(* IEC 61131-3 sources: SmartHomeNew/snapshots/2026-05-05 (part 2) *)

(* ---- PRG_IO_Write.st ---- *)
PROGRAM PRG_IO_Write
VAR
    L_i : INT;
    L_Heating_Forced_Off : BOOL;
    L_Vent_Forced_Off : BOOL;
    L_Water_Forced_Off : BOOL;
    L_Access_Forced_Off : BOOL;
    L_Access_Safety_Override : BOOL;
    L_Global_Hard_Stop : BOOL;
    L_Gas_Safety_Stop : BOOL;
    L_Freeze_Active : BOOL;
    L_Gas_Fire_Siren_Enable : BOOL;
    fbTrace : FB_Trace_Write;
END_VAR

L_Global_Hard_Stop := GVL_COMMAND_SHADOW.G_Heating_Emergency_Stop;
L_Gas_Safety_Stop := GVL_COMMAND_SHADOW.G_Heating_Gas_Safety_Stop OR GVL_COMMAND_SHADOW.G_Boiler_Stop;
L_Freeze_Active := GVL_STATE.G_Safety_Freeze_Risk;
L_Gas_Fire_Siren_Enable := GVL_ALARM.G_Gas_Fire_Siren OR GVL_ALARM.G_Global_Siren OR GVL_ALARM.G_Global_Critical;

IF NOT GVL_STATUS.G_Is_Active_PLC OR L_Global_Hard_Stop THEN
    FOR L_i := 1 TO GVL_CONSTANTS.C_MAX_HEATING_CIRCUITS DO GVL_IO.DO_Zone_Valves[L_i] := FALSE; END_FOR;
    FOR L_i := 1 TO GVL_CONSTANTS.C_MAX_MANIFOLDS DO GVL_IO.DO_Manifold_Pumps[L_i] := FALSE; GVL_IO.AO_Manifold_Valves[L_i] := 0; END_FOR;
    GVL_IO.DO_DHW_Heating_Pump := FALSE;
    GVL_IO.DO_DHW_Circ_Pump := FALSE;
    GVL_IO.DO_Backup_Circulation_Pump := FALSE;
    GVL_IO.DO_Electric_Heater_Enable := FALSE;
    FOR L_i := 1 TO GVL_CONSTANTS.C_MAX_SUPPLY_FANS DO GVL_IO.AO_Supply_Fans[L_i] := 0; END_FOR;
    FOR L_i := 1 TO GVL_CONSTANTS.C_MAX_EXHAUST_FANS DO GVL_IO.AO_Exhaust_Fans[L_i] := 0; END_FOR;
    FOR L_i := 1 TO GVL_CONSTANTS.C_MAX_WATER_ZONES DO GVL_IO.DO_Water_Zone_Enable[L_i] := FALSE; END_FOR;
    FOR L_i := 1 TO GVL_CONSTANTS.C_MAX_LIGHT_ZONES DO GVL_IO.AO_Lighting_Levels[L_i] := 0; END_FOR;
    FOR L_i := 1 TO GVL_CONSTANTS.C_MAX_BLINDS DO GVL_IO.AO_Blinds_Positions[L_i] := 1000; END_FOR;
    FOR L_i := 1 TO GVL_CONSTANTS.C_MAX_SOCKETS DO GVL_IO.DO_Sockets[L_i] := FALSE; END_FOR;
    GVL_IO.DO_Gate_Open := FALSE;
    GVL_IO.DO_Wicket_Open := FALSE;
    GVL_IO.DO_Lock_1_Open := FALSE;
    GVL_IO.DO_Lock_1_Close := FALSE;
    GVL_IO.DO_Lock_2_Open := FALSE;
    GVL_IO.DO_Lock_2_Close := FALSE;
    GVL_IO.DO_Gas_Siren := L_Gas_Fire_Siren_Enable AND GVL_ALARM.G_Gas_Alarm_Active;
    GVL_IO.DO_Fire_Siren := L_Gas_Fire_Siren_Enable AND GVL_ALARM.G_Fire_Alarm_Active;
    GVL_IO.DO_Security_Siren := GVL_ALARM.G_Security_Siren OR (GVL_ALARM.G_Global_Siren AND GVL_ALARM.G_Security_Alarm);
    GVL_IO.DO_Gas_Valve_Close := TRUE;
    RETURN;
END_IF;

L_Heating_Forced_Off := GVL_COMMAND_SHADOW.G_Heating_Block;
L_Vent_Forced_Off := GVL_COMMAND_SHADOW.G_Vent_Stop OR GVL_COMMAND_SHADOW.G_Vent_Block;
L_Water_Forced_Off := GVL_COMMAND_SHADOW.G_Water_Block OR GVL_COMMAND_SHADOW.G_Water_Emergency_Stop;

L_Access_Safety_Override := (GVL_SAFETY_SHUTDOWN.G_Safety_Mode = FIRE) OR (GVL_SAFETY_SHUTDOWN.G_Safety_Mode = GAS);
L_Access_Forced_Off := GVL_SAFETY_RECOVERY.G_Recovery_Active AND NOT L_Access_Safety_Override;

FOR L_i := 1 TO GVL_CONSTANTS.C_MAX_HEATING_CIRCUITS DO
    IF (L_i > GVL_SYSTEM_SIZE_CONFIG.G_Active_Heating_Circuits) OR L_Heating_Forced_Off THEN
        GVL_IO.DO_Zone_Valves[L_i] := FALSE;
    ELSE
        GVL_IO.DO_Zone_Valves[L_i] := GVL_HEATING_OUTPUT.DO_Zone_Valves[L_i];
    END_IF;
END_FOR;

FOR L_i := 1 TO GVL_CONSTANTS.C_MAX_MANIFOLDS DO
    IF L_Heating_Forced_Off AND NOT (L_Gas_Safety_Stop AND L_Freeze_Active) THEN
        GVL_IO.DO_Manifold_Pumps[L_i] := FALSE;
        GVL_IO.AO_Manifold_Valves[L_i] := 0;
    ELSE
        GVL_IO.DO_Manifold_Pumps[L_i] := GVL_HEATING_OUTPUT.DO_Manifold_Pumps[L_i];
        GVL_IO.AO_Manifold_Valves[L_i] := GVL_HEATING_OUTPUT.AO_Manifold_Valves[L_i];
    END_IF;
END_FOR;

IF L_Heating_Forced_Off AND NOT (L_Gas_Safety_Stop AND L_Freeze_Active) THEN
    GVL_IO.DO_DHW_Heating_Pump := FALSE;
    GVL_IO.DO_DHW_Circ_Pump := FALSE;
    GVL_IO.DO_Backup_Circulation_Pump := FALSE;
    GVL_IO.DO_Electric_Heater_Enable := FALSE;
ELSE
    GVL_IO.DO_DHW_Heating_Pump := FALSE;
    GVL_IO.DO_DHW_Circ_Pump := GVL_HEATING_OUTPUT.DO_DHW_Circ_Pump;
    GVL_IO.DO_Backup_Circulation_Pump := GVL_HEATING_OUTPUT.DO_Backup_Circulation_Pump;
    GVL_IO.DO_Electric_Heater_Enable := GVL_HEATING_OUTPUT.DO_Electric_Heater_Enable;
END_IF;

FOR L_i := 1 TO GVL_CONSTANTS.C_MAX_SUPPLY_FANS DO
    IF L_Vent_Forced_Off THEN
        GVL_IO.AO_Supply_Fans[L_i] := 0;
    ELSE
        GVL_IO.AO_Supply_Fans[L_i] := GVL_VENT_OUTPUT.AO_Supply_Fans[L_i];
    END_IF;
END_FOR;

FOR L_i := 1 TO GVL_CONSTANTS.C_MAX_EXHAUST_FANS DO
    IF L_Vent_Forced_Off THEN
        GVL_IO.AO_Exhaust_Fans[L_i] := 0;
    ELSE
        GVL_IO.AO_Exhaust_Fans[L_i] := GVL_VENT_OUTPUT.AO_Exhaust_Fans[L_i];
    END_IF;
END_FOR;

// FIXED: water valves now from domain output
GVL_IO.DO_Water_Valve_35_Close := GVL_WATER_OUTPUT.DO_Water_Valve_35_Close;
GVL_IO.DO_Water_Valve_36_Close := GVL_WATER_OUTPUT.DO_Water_Valve_36_Close;

FOR L_i := 1 TO GVL_CONSTANTS.C_MAX_WATER_ZONES DO
    IF (L_i > GVL_SYSTEM_SIZE_CONFIG.G_Active_Water_Zones) OR L_Water_Forced_Off THEN
        GVL_IO.DO_Water_Zone_Enable[L_i] := FALSE;
    ELSE
        GVL_IO.DO_Water_Zone_Enable[L_i] := GVL_WATER_OUTPUT.DO_Water_Zone_Enable[L_i];
    END_IF;
END_FOR;

FOR L_i := 1 TO GVL_CONSTANTS.C_MAX_LIGHT_ZONES DO
    GVL_IO.AO_Lighting_Levels[L_i] := BYTE_TO_UINT(GVL_STATE.G_Lighting_Levels[L_i]) * 10;
END_FOR;

FOR L_i := 1 TO GVL_CONSTANTS.C_MAX_BLINDS DO
    GVL_IO.AO_Blinds_Positions[L_i] := BYTE_TO_UINT(GVL_STATE.G_Blinds_Positions[L_i]) * 10;
END_FOR;

FOR L_i := 1 TO GVL_CONSTANTS.C_MAX_SOCKETS DO
    GVL_IO.DO_Sockets[L_i] := GVL_STATE.G_Socket_States[L_i];
END_FOR;

IF L_Access_Forced_Off THEN
    GVL_IO.DO_Gate_Open := FALSE;
    GVL_IO.DO_Wicket_Open := FALSE;
    GVL_IO.DO_Lock_1_Open := FALSE;
    GVL_IO.DO_Lock_1_Close := FALSE;
    GVL_IO.DO_Lock_2_Open := FALSE;
    GVL_IO.DO_Lock_2_Close := FALSE;
ELSE
    GVL_IO.DO_Gate_Open := GVL_ACCESS_OUTPUT.DO_Gate_Open;
    GVL_IO.DO_Wicket_Open := GVL_ACCESS_OUTPUT.DO_Wicket_Open;
    GVL_IO.DO_Lock_1_Open := GVL_ACCESS_OUTPUT.DO_Lock_1_Open;
    GVL_IO.DO_Lock_1_Close := GVL_ACCESS_OUTPUT.DO_Lock_1_Close;
    GVL_IO.DO_Lock_2_Open := GVL_ACCESS_OUTPUT.DO_Lock_2_Open;
    GVL_IO.DO_Lock_2_Close := GVL_ACCESS_OUTPUT.DO_Lock_2_Close;
END_IF;

GVL_IO.DO_Gas_Siren := L_Gas_Fire_Siren_Enable AND GVL_ALARM.G_Gas_Alarm_Active;
GVL_IO.DO_Fire_Siren := L_Gas_Fire_Siren_Enable AND GVL_ALARM.G_Fire_Alarm_Active;
GVL_IO.DO_Security_Siren := GVL_ALARM.G_Security_Siren OR (GVL_ALARM.G_Global_Siren AND GVL_ALARM.G_Security_Alarm);
GVL_IO.DO_Gas_Valve_Close := GVL_COMMAND_SHADOW.G_Gas_Valve_Close;

fbTrace(iLayer := TRACE_IO,iSource := SRC_IO,iReason := REASON_DOMAIN_PROJECTION,iValueBool := TRUE,iValueReal := 0.0,iText := 'IO write projection executed');
END_PROGRAM

(* ---- PRG_Presence_Manager.st ---- *)
PROGRAM PRG_Presence_Manager
VAR
    fbPresence : FB_Presence_Manager;
    L_i : INT;
END_VAR

fbPresence(
    VI_Motion_Sensors := GVL_STATE.G_Motion_Sensors,
    VI_System_Time_MS := GVL_STATUS.G_System_Time_MS
);

GVL_PRESENCE.G_Any_Motion := fbPresence.VO_Any_Motion;
GVL_PRESENCE.G_Occupied := fbPresence.VO_Occupied;
GVL_PRESENCE.G_Auto_Away_Request := fbPresence.VO_Auto_Away;
GVL_PRESENCE.G_Last_Motion_TS := fbPresence.VO_Last_Motion_TS;

FOR L_i := 1 TO GVL_CONSTANTS.C_MAX_ZONES DO
    IF GVL_STATE.G_Motion_Sensors[L_i] THEN
        GVL_PRESENCE.G_Zone_Occupied[L_i] := TRUE;
        GVL_PRESENCE.G_Zone_Last_Motion_TS[L_i] := GVL_STATUS.G_System_Time_MS;
    END_IF;

    IF (GVL_STATUS.G_System_Time_MS - GVL_PRESENCE.G_Zone_Last_Motion_TS[L_i]) > 900000 THEN
        GVL_PRESENCE.G_Zone_Occupied[L_i] := FALSE;
    END_IF;
END_FOR;
END_PROGRAM

(* ---- PRG_Safety_Recovery.st ---- *)
PROGRAM PRG_Safety_Recovery
VAR
    L_Phase : E_Recovery_Phase;
    L_Mode_Active : BOOL;
    L_Time_OK : BOOL;
END_VAR

L_Mode_Active := GVL_SAFETY_SHUTDOWN.G_Safety_Active;
L_Phase := GVL_SAFETY_RECOVERY.G_Recovery_Phase;

CASE L_Phase OF

    IDLE:
        IF NOT L_Mode_Active AND GVL_SAFETY_RECOVERY.G_Recovery_Requested THEN
            GVL_SAFETY_RECOVERY.G_Recovery_Phase := STABILIZING;
            GVL_SAFETY_RECOVERY.G_Recovery_Active := TRUE;
            GVL_SAFETY_RECOVERY.G_Recovery_Start_MS := GVL_TIME_SERVICE.G_Now_MS;
        END_IF;

    STABILIZING:
        IF L_Mode_Active THEN
            GVL_SAFETY_RECOVERY.G_Recovery_Phase := ABORTED;
            GVL_SAFETY_RECOVERY.G_Recovery_Abort_Reason := 1;
        ELSIF (GVL_TIME_SERVICE.G_Now_MS - GVL_SAFETY_RECOVERY.G_Recovery_Start_MS) > GVL_SAFETY_RECOVERY_CONFIG.G_Stabilization_Delay_MS THEN
            GVL_SAFETY_RECOVERY.G_Recovery_Phase := WAIT_MANUAL_CONFIRM;
            GVL_SAFETY_RECOVERY.G_Recovery_Stable_Since_MS := GVL_TIME_SERVICE.G_Now_MS;
        END_IF;

    WAIT_MANUAL_CONFIRM:
        IF L_Mode_Active THEN
            GVL_SAFETY_RECOVERY.G_Recovery_Phase := ABORTED;
            GVL_SAFETY_RECOVERY.G_Recovery_Abort_Reason := 1;
        ELSIF GVL_SAFETY_RECOVERY.G_Recovery_Manual_Confirm THEN
            GVL_SAFETY_RECOVERY.G_Recovery_Phase := RECOVERING;
        END_IF;

    RECOVERING:
        IF L_Mode_Active THEN
            GVL_SAFETY_RECOVERY.G_Recovery_Phase := ABORTED;
            GVL_SAFETY_RECOVERY.G_Recovery_Abort_Reason := 1;
        ELSE
            GVL_SAFETY_RECOVERY.G_Recovery_Phase := COOLDOWN;
            GVL_SAFETY_RECOVERY.G_Recovery_Cooldown_Start_MS := GVL_TIME_SERVICE.G_Now_MS;
        END_IF;

    COOLDOWN:
        IF L_Mode_Active THEN
            GVL_SAFETY_RECOVERY.G_Recovery_Phase := ABORTED;
            GVL_SAFETY_RECOVERY.G_Recovery_Abort_Reason := 1;
        ELSE
            L_Time_OK := (GVL_TIME_SERVICE.G_Now_MS - GVL_SAFETY_RECOVERY.G_Recovery_Cooldown_Start_MS) > GVL_SAFETY_RECOVERY_CONFIG.G_Cooldown_Time_MS;

            IF L_Time_OK THEN
                GVL_SAFETY_RECOVERY.G_Recovery_Phase := IDLE;
                GVL_SAFETY_RECOVERY.G_Recovery_Active := FALSE;
                GVL_SAFETY_RECOVERY.G_Recovery_Requested := FALSE;
                GVL_SAFETY_RECOVERY.G_Recovery_Manual_Confirm := FALSE;
            END_IF;
        END_IF;

    ABORTED:
        GVL_SAFETY_RECOVERY.G_Recovery_Active := FALSE;
        IF NOT L_Mode_Active THEN
            GVL_SAFETY_RECOVERY.G_Recovery_Phase := IDLE;
        END_IF;

END_CASE;

END_PROGRAM
// >>> BULK_SYNC_ANCHOR: PRG_Safety_Recovery <<<

(* ---- PRG_System_Alarm_Gateway.st ---- *)
PROGRAM PRG_System_Alarm_Gateway
VAR
    fbSystemAlarmOrchestrator : FB_System_Alarm_Orchestrator;
    fbSystemGatewayIntent : FB_System_Gateway_Intent;
    L_Scenario_Req_Gateway : E_SCENARIO_TYPE;
END_VAR

// Alarm orchestration based on global health snapshot
fbSystemAlarmOrchestrator(
    VI_First_Fault_Active := GVL_SYSTEM_HEALTH.G_First_Fault_Active,
    VI_First_Fault_Type := GVL_SYSTEM_HEALTH.G_First_Fault_Type,
    VI_First_Fault_Source := GVL_SYSTEM_HEALTH.G_First_Fault_Source
);

// Gateway intent execution
fbSystemGatewayIntent(
    VI_System_Time_MS := GVL_TIME_SERVICE.G_Now_MS,
    VI_IsActivePLC := GVL_STATUS.G_Is_Active_PLC,
    VI_Gateway_Writes_Allowed := NOT GVL_STATUS.G_Diagnostics.Operator_Action_Blocked,
    VIO_FloorHeating_Temps := GVL_STATE.G_Floor_Temps,
    VIO_Zone_Valve_States := GVL_STATE.G_Zone_Valves,
    VIO_Lighting_Base_Levels := GVL_STATE.G_Lighting_Levels,
    VIO_Scenario_Req_Gateway := L_Scenario_Req_Gateway
);

GVL_INTENT_USER.I_Scenario_Request := L_Scenario_Req_Gateway;

END_PROGRAM
